FUNCTION_BLOCK WagoDistributingStation (* Composite Function Block Type *)
  (* Standard: 61499-2 *)
  (* Version 0.2, 2003-12-05, JHC, Rockwell Automation, Renamed from NEWCOMPFB. *)
  (* Compiler header: package fb.rt.wago; *)
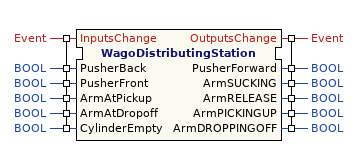
  EVENT_INPUT
    InputsChange WITH PusherBack, PusherFront, ArmAtPickup, ArmAtDropoff, CylinderEmpty;
  END_EVENT
  EVENT_OUTPUT
    OutputsChange WITH PusherAtBack, PusherForward, ArmPICKINGUP, ArmDROPPINGOFF, ArmSUCKING, ArmRELEASE;
  END_EVENT
  VAR_INPUT
    PusherBack : BOOL; (* Input event qualifier *)
    PusherFront : BOOL; (* Input event qualifier *)
    ArmAtPickup : BOOL; (* Input event qualifier *)
    ArmAtDropoff : BOOL; (* Input event qualifier *)
    CylinderEmpty : BOOL; (* Input event qualifier *)
  END_VAR
  VAR_OUTPUT
    PusherForward : BOOL := false;
    ArmSUCKING : BOOL := false;
    ArmRELEASE : BOOL := false;
    ArmPICKINGUP : BOOL := false;
    ArmDROPPINGOFF : BOOL := false; (* Output event qualifier *)
  END_VAR
  FBS
    DistStnArm : DistStnArm;
    DistStnPusher : DistStnPusher;
  END_FBS
  EVENT_CONNECTIONS
    InputsChange TO DistStnPusher.PosChange;
    InputsChange TO DistStnArm.PosChange;
    DistStnArm.ArmCtrl TO OutputsChange;
    DistStnPusher.PusherCtrl TO OutputsChange;
    DistStnPusher.ItemStatus TO DistStnArm.ItemStatus;
    DistStnArm.ArmStatus TO DistStnPusher.ArmStatusChange;
  END_CONNECTIONS
  DATA_CONNECTIONS
    PusherBack TO DistStnPusher.PosBack;
    PusherFront TO DistStnPusher.PosFront;
    CylinderEmpty TO DistStnPusher.CylinderEmpty;
    ArmAtPickup TO DistStnArm.PosReadyToSuck;
    ArmAtDropoff TO DistStnArm.PosReadyToDrop;
    DistStnArm.ArmPICKINGUP TO ArmPICKINGUP;
    DistStnArm.ArmDROPPINGOFF TO ArmDROPPINGOFF;
    DistStnArm.ArmSUCKING TO ArmSUCKING;
    DistStnArm.ArmRELEASE TO ArmRELEASE;
    DistStnPusher.PusherForward TO PusherForward;
    DistStnPusher.ItemPresent TO DistStnArm.ItemNeedingPickup;
    DistStnArm.ArmClear TO DistStnPusher.ArmClear;
  END_CONNECTIONS
END_FUNCTION_BLOCK
